{attribute 'no_explicit_call' := 'do not call this POU directly'} 
FUNCTION_BLOCK AnalogInput IMPLEMENTS I_AnalogChannel
VAR_INPUT
END_VAR
VAR_OUTPUT
END_VAR
VAR
    {attribute 'TcInitSymbol'}
	ID:				STRING(25);	// Equipment ID
	Channel			AT%I*: INT;
END_VAR

PROPERTY PUBLIC P_ID : String(25)
GET
P_ID:= ID;
END_GET
END_PROPERTY

PROPERTY P_State : EPlcMappingStatus
GET
P_State:= F_GetMappingStatus(ADR(Channel), SIZEOF(INT));
END_GET
END_PROPERTY

PROPERTY PUBLIC P_Value : Lreal
GET
P_Value:= INT_TO_LREAL(Channel);
END_GET
SET // PUBLIC
Channel:= LREAL_TO_INT(P_Value);
END_SET
END_PROPERTY

END_FUNCTION_BLOCK

(* stored: Version 1.1.0.1
   POU AnalogInput: Id {4b790aa2-3d71-03d0-3f43-731f51993f5b}, SpecialFunc None
   Property P_ID: Id {a66b090d-1b03-0814-2c19-26bfc0a32879}
   Get Get: Id {fc6b929d-a455-0724-220a-60cfdcf325e2}
   Property P_State: Id {5cd81f9d-9d09-0ac9-22c0-8458e557abfb}
   Get Get: Id {550aa5b6-4e2e-02eb-086b-4a4d1283c230}
   Property P_Value: Id {f773b0b4-8cc1-09cc-39ec-af3ba89db27d}
   Get Get: Id {20aacbb5-6c42-0d45-142f-45cfd18fd613}
   Set Set: Id {9ddffbf9-2bf0-046e-0e43-6682be3f435e} *)
